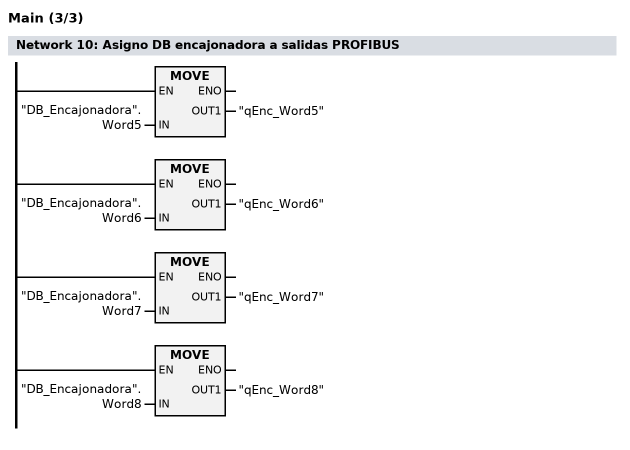
   RUNG wire#powerrail
      Move(in := "DB_Encajonadora".Word5, out1 => "qEnc_Word5")
   END_RUNG
   RUNG wire#powerrail
      Move(in := "DB_Encajonadora".Word6, out1 => "qEnc_Word6")
   END_RUNG
   RUNG wire#powerrail
      Move(in := "DB_Encajonadora".Word7, out1 => "qEnc_Word7")
   END_RUNG
   RUNG wire#powerrail
      Move(in := "DB_Encajonadora".Word8, out1 => "qEnc_Word8")
   END_RUNG
   // the same network as SCL:
   "qEnc_Word5" := "DB_Encajonadora".Word5;
   "qEnc_Word6" := "DB_Encajonadora".Word6;
   "qEnc_Word7" := "DB_Encajonadora".Word7;
   "qEnc_Word8" := "DB_Encajonadora".Word8;
END_REGION
END_ORGANIZATION_BLOCK

ORGANIZATION_BLOCK "Cyclic interrupt"   // OB30, LAD, CyclicInterrupt
{ S7_Optimized_Access := 'TRUE' }
VERSION : 0.1
   VAR_INPUT
      Initial_Call : Bool;   // Initial call of this OB
      Event_Count : Int;   // Events discarded
   END_VAR
BEGIN

REGION Network 1: Move
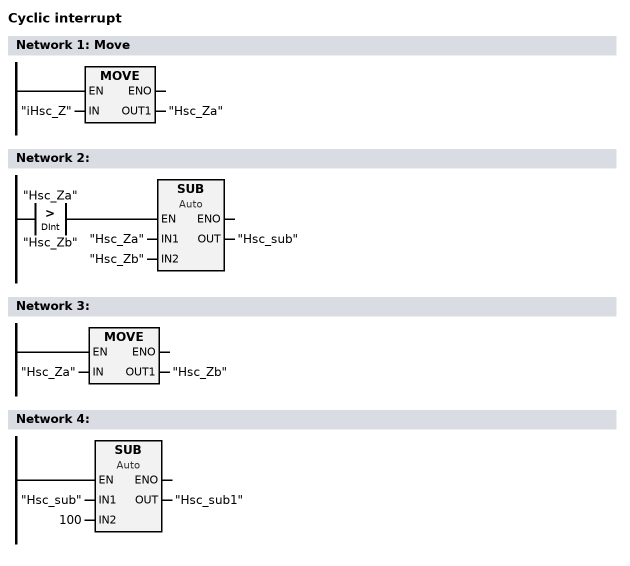
   RUNG wire#powerrail
      Move(in := "iHsc_Z", out1 => "Hsc_Za")
   END_RUNG
   // the same network as SCL:
   "Hsc_Za" := "iHsc_Z";
END_REGION

REGION Network 2
   RUNG wire#powerrail
      { S7_Templates := "SrcType := DInt" } GT_Contact(in1 := "Hsc_Za", in2 := "Hsc_Zb")
      Sub(in1 := "Hsc_Za", in2 := "Hsc_Zb", out => "Hsc_sub")
   END_RUNG
   // the same network as SCL:
   IF "Hsc_Za" > "Hsc_Zb" THEN "Hsc_sub" := "Hsc_Za" - "Hsc_Zb"; END_IF;
END_REGION

REGION Network 3
   RUNG wire#powerrail
      Move(in := "Hsc_Za", out1 => "Hsc_Zb")
   END_RUNG
   // the same network as SCL:
   "Hsc_Zb" := "Hsc_Za";
END_REGION

REGION Network 4
   RUNG wire#powerrail
      Sub(in1 := "Hsc_sub", in2 := 100, out => "Hsc_sub1")
   END_RUNG
   // the same network as SCL:
   "Hsc_sub1" := "Hsc_sub" - 100;
END_REGION
END_ORGANIZATION_BLOCK

// folder: ESTANDAR

FUNCTION_BLOCK "Motor M&CM"   // FB2, LAD
TITLE = Motor Marcha & Contra-Marcha
{ S7_Optimized_Access := 'TRUE' }
VERSION : 0.1
   VAR_INPUT
      iOrdMar_Dir : Bool;
      iOrdMar_Rev : Bool;
      iConfMar_Dir : Bool;
      iConfMar_Rev : Bool;
      iGMT : Bool;
      iTConf_Warn : Time;
      iTConf_Fall : Time;
      iTRearranque : Time;
   END_VAR
   VAR_OUTPUT
      oMar_Dir : Bool;
      oMar_Rev : Bool;
      oWarning_CTC_Dir : Bool;
      oWarning_CTC_Rev : Bool;
      oFall_CTC_Dir : Bool;
      oFall_CTC_Rev : Bool;
      oFall_GMT : Bool;
   END_VAR
   VAR
      IEC_Timer_0_Instance : IEC_TIMER;
      IEC_Timer_0_Instance_1 : IEC_TIMER;
      IEC_Timer_0_Instance_2 : IEC_TIMER;
      IEC_Timer_0_Instance_3 : IEC_TIMER;
      IEC_Timer_0_Instance_4 : IEC_TIMER;
      MarDir_Aux : Bool;
      MarRev_Aux : Bool;
   END_VAR
   VAR_TEMP
      Fall_GMT_Aux : Bool;
      Fall_CTC_Dir_Aux : Bool;
      Fall_CTC_Rev_Aux : Bool;
      Habil_Mov : Bool;
   END_VAR
   VAR_TEMP   // added for the SCL form of the ladder/FBD networks
      _w1 : Bool;
   END_VAR
BEGIN

REGION Network 1: Falla Guardamotor
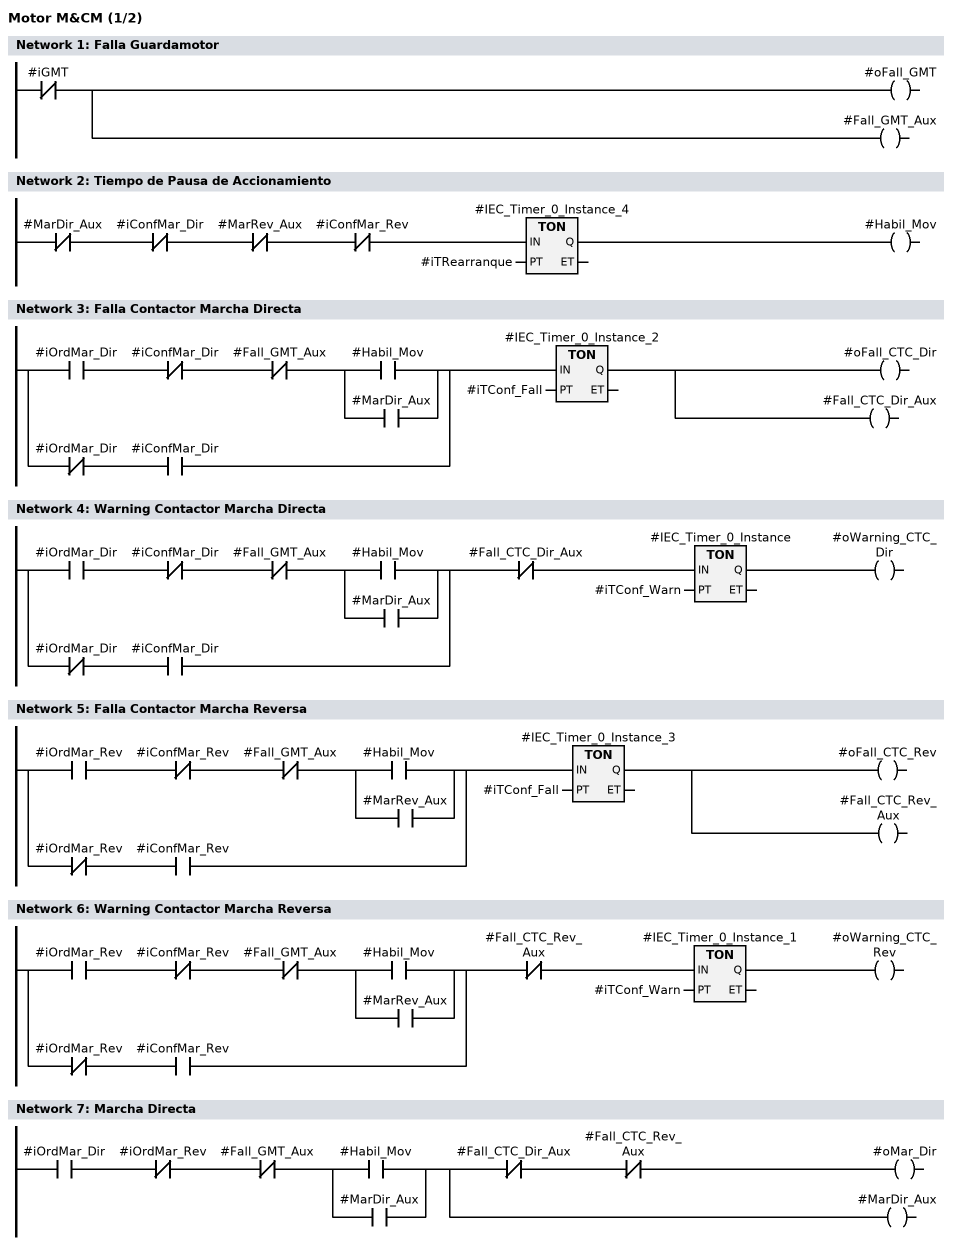
   RUNG wire#powerrail
      I_Contact( #iGMT )
      wire#w1
      Coil( #oFall_GMT )
   END_RUNG
   RUNG wire#w1
      Coil( #Fall_GMT_Aux )
   END_RUNG
   // the same network as SCL:
   #oFall_GMT := NOT #iGMT;
   #Fall_GMT_Aux := NOT #iGMT;
END_REGION

REGION Network 2: Tiempo de Pausa de Accionamiento
   #IEC_Timer_0_Instance_4.TON(IN := NOT #MarDir_Aux AND NOT #iConfMar_Dir AND NOT #MarRev_Aux AND NOT #iConfMar_Rev,
                           PT := #iTRearranque);
   #Habil_Mov := #IEC_Timer_0_Instance_4.Q;
END_REGION

REGION Network 3: Falla Contactor Marcha Directa
   #IEC_Timer_0_Instance_2.TON(IN := (#iOrdMar_Dir AND NOT #iConfMar_Dir AND NOT #Fall_GMT_Aux AND (#Habil_Mov OR #MarDir_Aux)) OR (NOT #iOrdMar_Dir AND #iConfMar_Dir),
                           PT := #iTConf_Fall);
   #oFall_CTC_Dir := #IEC_Timer_0_Instance_2.Q;
   #Fall_CTC_Dir_Aux := #IEC_Timer_0_Instance_2.Q;
END_REGION

REGION Network 4: Warning Contactor Marcha Directa
   #IEC_Timer_0_Instance.TON(IN := ((#iOrdMar_Dir AND NOT #iConfMar_Dir AND NOT #Fall_GMT_Aux AND (#Habil_Mov OR #MarDir_Aux)) OR (NOT #iOrdMar_Dir AND #iConfMar_Dir)) AND NOT #Fall_CTC_Dir_Aux,
                           PT := #iTConf_Warn);
   #oWarning_CTC_Dir := #IEC_Timer_0_Instance.Q;
END_REGION

REGION Network 5: Falla Contactor Marcha Reversa
   #IEC_Timer_0_Instance_3.TON(IN := (#iOrdMar_Rev AND NOT #iConfMar_Rev AND NOT #Fall_GMT_Aux AND (#Habil_Mov OR #MarRev_Aux)) OR (NOT #iOrdMar_Rev AND #iConfMar_Rev),
                           PT := #iTConf_Fall);
   #oFall_CTC_Rev := #IEC_Timer_0_Instance_3.Q;
   #Fall_CTC_Rev_Aux := #IEC_Timer_0_Instance_3.Q;
END_REGION

REGION Network 6: Warning Contactor Marcha Reversa
   #IEC_Timer_0_Instance_1.TON(IN := ((#iOrdMar_Rev AND NOT #iConfMar_Rev AND NOT #Fall_GMT_Aux AND (#Habil_Mov OR #MarRev_Aux)) OR (NOT #iOrdMar_Rev AND #iConfMar_Rev)) AND NOT #Fall_CTC_Rev_Aux,
                           PT := #iTConf_Warn);
   #oWarning_CTC_Rev := #IEC_Timer_0_Instance_1.Q;
END_REGION

REGION Network 7: Marcha Directa
   RUNG wire#powerrail
      Contact( #iOrdMar_Dir )
      I_Contact( #iOrdMar_Rev )
      I_Contact( #Fall_GMT_Aux )
      wire#w1
      Contact( #Habil_Mov )
      wire#w2
      I_Contact( #Fall_CTC_Dir_Aux )
      I_Contact( #Fall_CTC_Rev_Aux )
      Coil( #oMar_Dir )
   END_RUNG
   RUNG wire#w1
      Contact( #MarDir_Aux )
   END_RUNG wire#w2
   RUNG wire#w2
      Coil( #MarDir_Aux )
   END_RUNG
   // the same network as SCL:
   #_w1 := #iOrdMar_Dir AND NOT #iOrdMar_Rev AND NOT #Fall_GMT_Aux AND (#Habil_Mov OR #MarDir_Aux);
   #oMar_Dir := #_w1 AND NOT #Fall_CTC_Dir_Aux AND NOT #Fall_CTC_Rev_Aux;
   #MarDir_Aux := #_w1;
END_REGION

REGION Network 8: Marcha Reversa
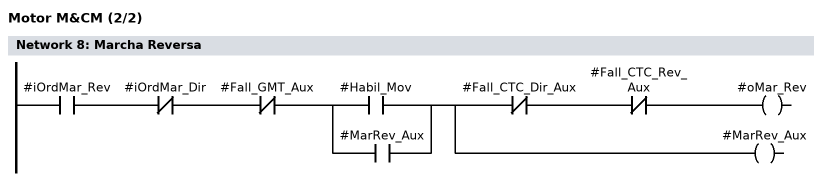
   RUNG wire#powerrail
      Contact( #iOrdMar_Rev )
      I_Contact( #iOrdMar_Dir )
      I_Contact( #Fall_GMT_Aux )
      wire#w1
      Contact( #Habil_Mov )
      wire#w2
      I_Contact( #Fall_CTC_Dir_Aux )
      I_Contact( #Fall_CTC_Rev_Aux )
      Coil( #oMar_Rev )
   END_RUNG
   RUNG wire#w1
      Contact( #MarRev_Aux )
   END_RUNG wire#w2
   RUNG wire#w2
      Coil( #MarRev_Aux )
   END_RUNG
   // the same network as SCL:
   #_w1 := #iOrdMar_Rev AND NOT #iOrdMar_Dir AND NOT #Fall_GMT_Aux AND (#Habil_Mov OR #MarRev_Aux);
   #oMar_Rev := #_w1 AND NOT #Fall_CTC_Dir_Aux AND NOT #Fall_CTC_Rev_Aux;
   #MarRev_Aux := #_w1;
END_REGION
END_FUNCTION_BLOCK

FUNCTION_BLOCK "FB_VAR_MOT"   // FB4, LAD
{ S7_Optimized_Access := 'FALSE' }
VERSION : 0.1
   VAR_INPUT
      "CMD Mar Dir" : Bool;   // Comando Marcha Directa
      "CMD Mar Rev" : Bool;   // Comando Marcha Reversa
      "HAB  Mar" : Bool;   // Habilita Marcha
      "SP Vel" : Real;   // Setpoint de Velocidad
      Reset : Bool;   // Comando resetear falla
      Fault : Bool;   // Indica variador en falla
      Ready : Bool;   // Indica variador Ready
      Ton_Freno : Time := T#400ms;
      Ton_Mar : Time := T#100ms;
      Tof_Freno : Time := T#100ms;
      Tof_Mar : Time := T#200ms;
   END_VAR
   VAR_OUTPUT
      Marcha : Bool;   // Orden de marcha a variador
      "Inv Giro" : Bool;   // Orden de invertir sentido de giro a variador
      "Reset Fault" : Bool;   // Reset Fault a variador
      Velocidad : Word;   // Referencia de Velocidad a variador
      Freno : Bool;   // Apertura de Freno
      Falla : Bool;   // Indica falla del variador
      Warning : Bool;   // Indica variador no Ready
   END_VAR
   VAR
      IEC_Timer_Freno : TON_TIME;
      IEC_Timer_Motor : TON_TIME;
      IEC_Timer_Reset : TOF_TIME;
      "_CMD Marcha Dir" : Bool;
      "_CMD Marcha Rev" : Bool;
      _CMD_AbrirFreno : Bool;
      IEC_Timer_0_Instance : TON_TIME;
      IEC_Timer_0_Instance_1 : TOF_TIME;
      IEC_Timer_0_Instance_2 : TOF_TIME;
      Ord_Marcha : Bool;
      Mem_Inv : Bool;
   END_VAR
   VAR_TEMP
      Vel_Real : Real;
      Vel_Int : Int;
      _Hab_Abrir_Freno : Bool;
      "Pre Marcha" : Bool;
      Aux : Bool;
      Freno_Aux : Bool;
   END_VAR
   VAR_TEMP   // added for the SCL form of the ladder/FBD networks
      _w1 : Bool;
      _w2 : Bool;
      _w3 : Bool;
   END_VAR
BEGIN

REGION Network 1: #Aux
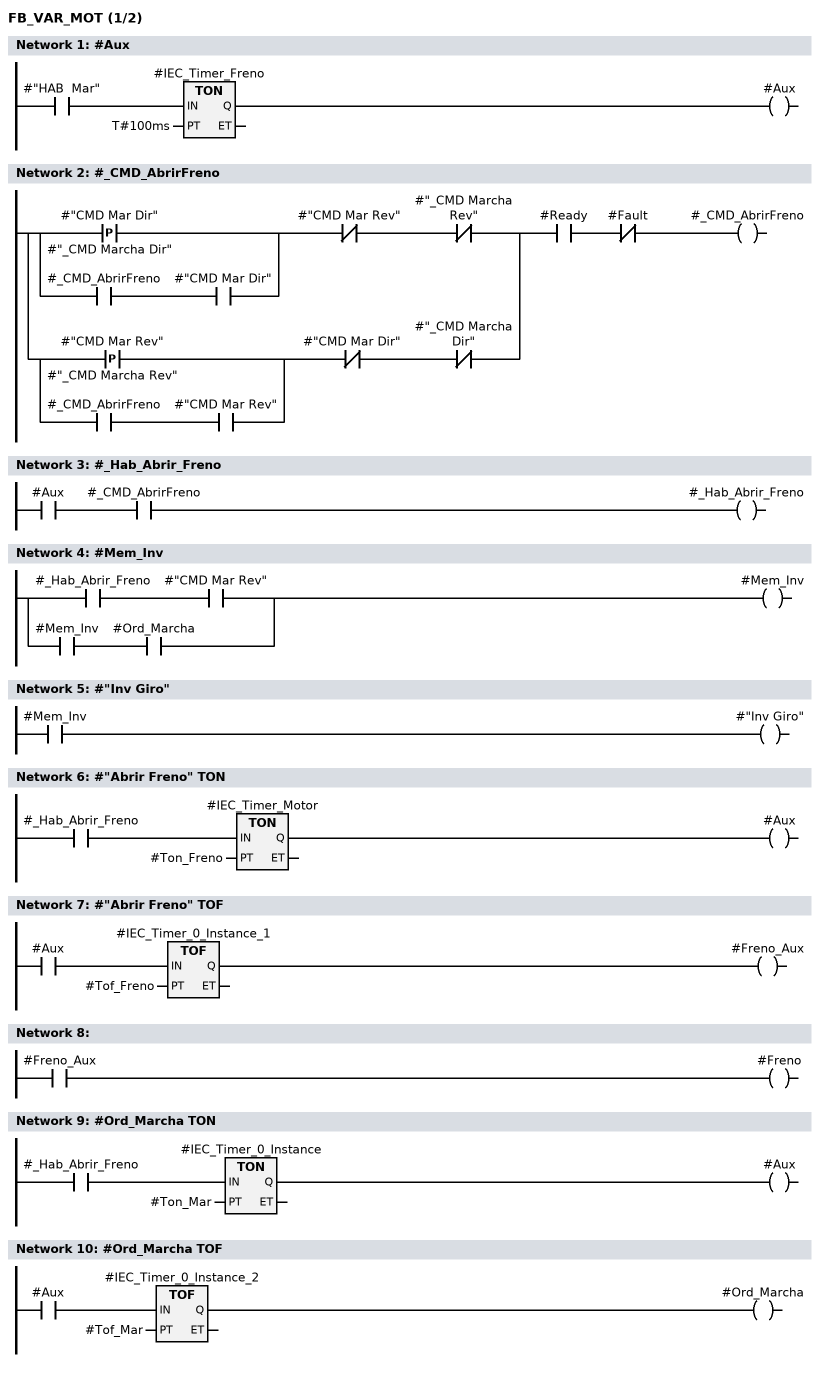
   #IEC_Timer_Freno(IN := #"HAB  Mar", PT := T#100ms);   // TON
   #Aux := #IEC_Timer_Freno.Q;
END_REGION

REGION Network 2: #_CMD_AbrirFreno
   RUNG wire#powerrail
      P_Contact(operand := #"CMD Mar Dir", bit := #"_CMD Marcha Dir")
      wire#w1
      I_Contact( #"CMD Mar Rev" )
      I_Contact( #"_CMD Marcha Rev" )
      wire#w2
      Contact( #Ready )
      I_Contact( #Fault )
      Coil( #_CMD_AbrirFreno )
   END_RUNG
   RUNG wire#powerrail
      Contact( #_CMD_AbrirFreno )
      Contact( #"CMD Mar Dir" )
   END_RUNG wire#w1
   RUNG wire#powerrail
      P_Contact(operand := #"CMD Mar Rev", bit := #"_CMD Marcha Rev")
      wire#w3
      I_Contact( #"CMD Mar Dir" )
      I_Contact( #"_CMD Marcha Dir" )
   END_RUNG wire#w2
   RUNG wire#powerrail
      Contact( #_CMD_AbrirFreno )
      Contact( #"CMD Mar Rev" )
   END_RUNG wire#w3
   // the same network as SCL:
   #_w1 := #"CMD Mar Dir" AND NOT #"_CMD Marcha Dir";   // rising edge of #"CMD Mar Dir"
   #"_CMD Marcha Dir" := #"CMD Mar Dir";
   #_w3 := (#_w1 OR (#_CMD_AbrirFreno AND #"CMD Mar Dir")) AND NOT #"CMD Mar Rev" AND NOT #"_CMD Marcha Rev";
   #_w2 := #"CMD Mar Rev" AND NOT #"_CMD Marcha Rev";   // rising edge of #"CMD Mar Rev"
   #"_CMD Marcha Rev" := #"CMD Mar Rev";
   #_CMD_AbrirFreno := (#_w3 OR ((#_w2 OR (#_CMD_AbrirFreno AND #"CMD Mar Rev")) AND NOT #"CMD Mar Dir" AND NOT #"_CMD Marcha Dir")) AND #Ready AND NOT #Fault;
END_REGION

REGION Network 3: #_Hab_Abrir_Freno
   RUNG wire#powerrail
      Contact( #Aux )
      Contact( #_CMD_AbrirFreno )
      Coil( #_Hab_Abrir_Freno )
   END_RUNG
   // the same network as SCL:
   #_Hab_Abrir_Freno := #Aux AND #_CMD_AbrirFreno;
END_REGION

REGION Network 4: #Mem_Inv
   RUNG wire#powerrail
      Contact( #_Hab_Abrir_Freno )
      Contact( #"CMD Mar Rev" )
      wire#w1
      Coil( #Mem_Inv )
   END_RUNG
   RUNG wire#powerrail
      Contact( #Mem_Inv )
      Contact( #Ord_Marcha )
   END_RUNG wire#w1
   // the same network as SCL:
   #Mem_Inv := (#_Hab_Abrir_Freno AND #"CMD Mar Rev") OR (#Mem_Inv AND #Ord_Marcha);
END_REGION

REGION Network 5: #"Inv Giro"
   RUNG wire#powerrail
      Contact( #Mem_Inv )
      Coil( #"Inv Giro" )
   END_RUNG
   // the same network as SCL:
   #"Inv Giro" := #Mem_Inv;
END_REGION

REGION Network 6: #"Abrir Freno" TON
   #IEC_Timer_Motor(IN := #_Hab_Abrir_Freno, PT := #Ton_Freno);   // TON
   #Aux := #IEC_Timer_Motor.Q;
END_REGION

REGION Network 7: #"Abrir Freno" TOF
   #IEC_Timer_0_Instance_1(IN := #Aux, PT := #Tof_Freno);   // TOF
   #Freno_Aux := #IEC_Timer_0_Instance_1.Q;
END_REGION

REGION Network 8
   RUNG wire#powerrail
      Contact( #Freno_Aux )
      Coil( #Freno )
   END_RUNG
   // the same network as SCL:
   #Freno := #Freno_Aux;
END_REGION

REGION Network 9: #Ord_Marcha TON
   #IEC_Timer_0_Instance(IN := #_Hab_Abrir_Freno, PT := #Ton_Mar);   // TON
   #Aux := #IEC_Timer_0_Instance.Q;
END_REGION

REGION Network 10: #Ord_Marcha TOF
   #IEC_Timer_0_Instance_2(IN := #Aux, PT := #Tof_Mar);   // TOF
   #Ord_Marcha := #IEC_Timer_0_Instance_2.Q;
END_REGION

REGION Network 11: #Marcha
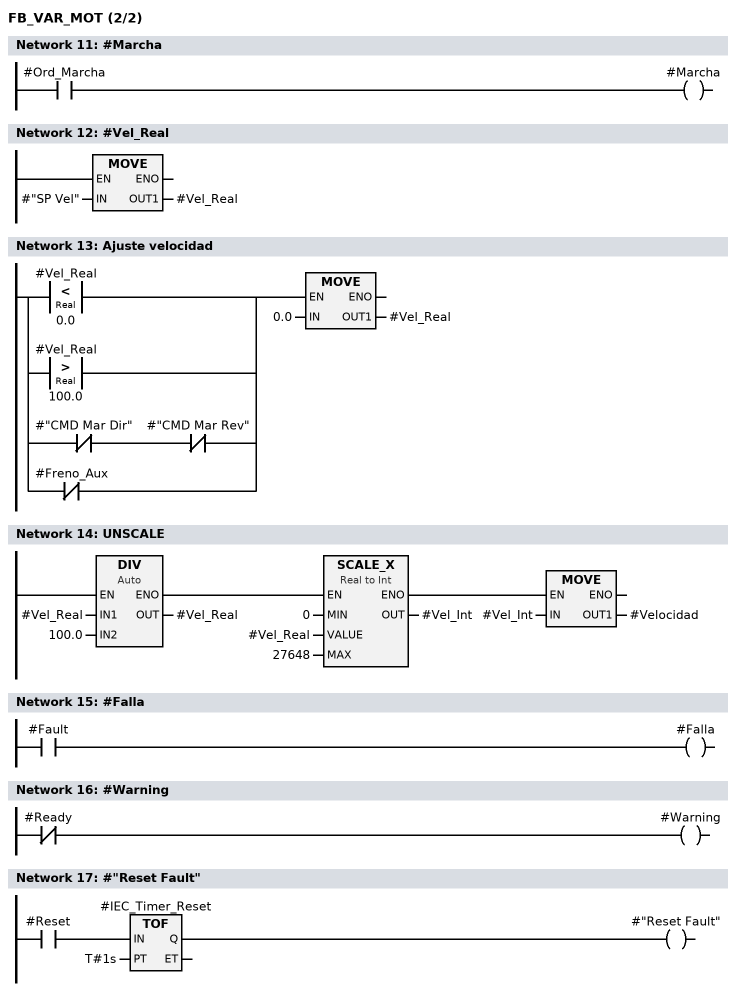
   RUNG wire#powerrail
      Contact( #Ord_Marcha )
      Coil( #Marcha )
   END_RUNG
   // the same network as SCL:
   #Marcha := #Ord_Marcha;
END_REGION

REGION Network 12: #Vel_Real
   RUNG wire#powerrail
      { S7_GenerateENO := "TRUE" } Move(in := #"SP Vel", out1 => #Vel_Real)
   END_RUNG
   // the same network as SCL:
   #Vel_Real := #"SP Vel";
END_REGION

REGION Network 13: Ajuste velocidad
   RUNG wire#powerrail
      { S7_Templates := "SrcType := Real" } LT_Contact(in1 := #Vel_Real, in2 := 0.0)
      wire#w1
      { S7_GenerateENO := "TRUE" } Move(in := 0.0, out1 => #Vel_Real)
   END_RUNG
   RUNG wire#powerrail
      { S7_Templates := "SrcType := Real" } GT_Contact(in1 := #Vel_Real, in2 := 100.0)
   END_RUNG wire#w1
   RUNG wire#powerrail
      I_Contact( #"CMD Mar Dir" )
      I_Contact( #"CMD Mar Rev" )
   END_RUNG wire#w1
   RUNG wire#powerrail
      I_Contact( #Freno_Aux )
   END_RUNG wire#w1
   // the same network as SCL:
   IF (#Vel_Real < 0.0) OR (#Vel_Real > 100.0) OR (NOT #"CMD Mar Dir" AND NOT #"CMD Mar Rev") OR NOT #Freno_Aux THEN
       #Vel_Real := 0.0;
   END_IF;
END_REGION

REGION Network 14: UNSCALE
   RUNG wire#powerrail
      Div(in1 := #Vel_Real, in2 := 100.0, out => #Vel_Real)
      { S7_Templates := "[SrcType := Real, DestType := Int]" } Scale(min := 0, value := #Vel_Real, max := 27648, out => #Vel_Int)
      { S7_GenerateENO := "TRUE" } Move(in := #Vel_Int, out1 => #Velocidad)
   END_RUNG
   // the same network as SCL:
   #Vel_Real := #Vel_Real / 100.0;
   #Vel_Int := SCALE_X(MIN := 0, VALUE := #Vel_Real, MAX := 27648);
   #Velocidad := #Vel_Int;
END_REGION

REGION Network 15: #Falla
   RUNG wire#powerrail
      Contact( #Fault )
      Coil( #Falla )
   END_RUNG
   // the same network as SCL:
   #Falla := #Fault;
END_REGION

REGION Network 16: #Warning
   RUNG wire#powerrail
      I_Contact( #Ready )
      Coil( #Warning )
   END_RUNG
   // the same network as SCL:
   #Warning := NOT #Ready;
END_REGION

REGION Network 17: #"Reset Fault"
   #IEC_Timer_Reset(IN := #Reset, PT := T#1s);   // TOF
   #"Reset Fault" := #IEC_Timer_Reset.Q;
END_REGION
END_FUNCTION_BLOCK

FUNCTION_BLOCK "Motor Simple"   // FB5, LAD
{ S7_Optimized_Access := 'TRUE' }
VERSION : 0.1
   VAR_INPUT
      iOrdMar : Bool;
      iConfMar : Bool;
      iGMT : Bool;
      iTConf_Warn : Time;
      iTConf_Fall : Time;
      iTRearranque : Time;
   END_VAR
   VAR_OUTPUT
      oMarcha : Bool;
      oWarning_CTC : Bool;
      oFall_CTC : Bool;
      oFall_GMT : Bool;
   END_VAR
   VAR
      IEC_Timer_0_Instance : IEC_TIMER;
      IEC_Timer_0_Instance_1 : IEC_TIMER;
      IEC_Timer_0_Instance_2 : IEC_TIMER;
      Mar_Aux : Bool;
   END_VAR
   VAR_TEMP
      Fall_GMT_Aux : Bool;
      Fall_CTC_Aux : Bool;
      Habil_Mov : Bool;
   END_VAR
BEGIN

REGION Network 1: Falla Guardamotor
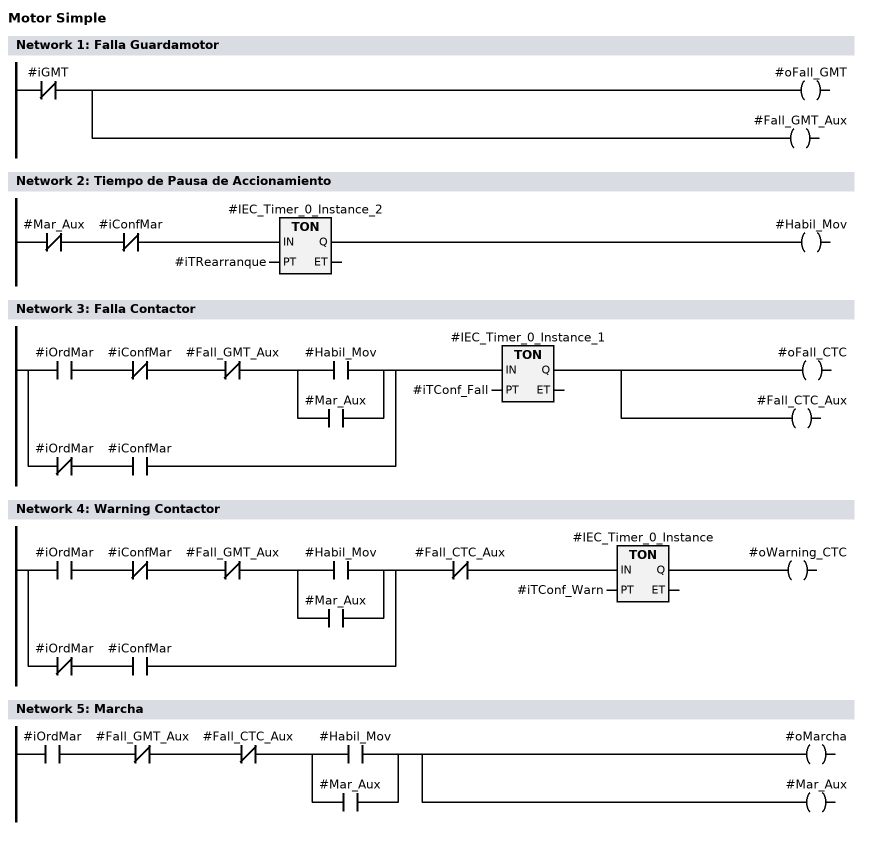
   RUNG wire#powerrail
      I_Contact( #iGMT )
      wire#w1
      Coil( #oFall_GMT )
   END_RUNG
   RUNG wire#w1
      Coil( #Fall_GMT_Aux )
   END_RUNG
   // the same network as SCL:
   #oFall_GMT := NOT #iGMT;
   #Fall_GMT_Aux := NOT #iGMT;
END_REGION

REGION Network 2: Tiempo de Pausa de Accionamiento
   #IEC_Timer_0_Instance_2.TON(IN := NOT #Mar_Aux AND NOT #iConfMar, PT := #iTRearranque);
   #Habil_Mov := #IEC_Timer_0_Instance_2.Q;
END_REGION

REGION Network 3: Falla Contactor
   #IEC_Timer_0_Instance_1.TON(IN := (#iOrdMar AND NOT #iConfMar AND NOT #Fall_GMT_Aux AND (#Habil_Mov OR #Mar_Aux)) OR (NOT #iOrdMar AND #iConfMar),
                           PT := #iTConf_Fall);
   #oFall_CTC := #IEC_Timer_0_Instance_1.Q;
   #Fall_CTC_Aux := #IEC_Timer_0_Instance_1.Q;
END_REGION

REGION Network 4: Warning Contactor
   #IEC_Timer_0_Instance.TON(IN := ((#iOrdMar AND NOT #iConfMar AND NOT #Fall_GMT_Aux AND (#Habil_Mov OR #Mar_Aux)) OR (NOT #iOrdMar AND #iConfMar)) AND NOT #Fall_CTC_Aux,
                           PT := #iTConf_Warn);
   #oWarning_CTC := #IEC_Timer_0_Instance.Q;
END_REGION

REGION Network 5: Marcha
   RUNG wire#powerrail
      Contact( #iOrdMar )
      I_Contact( #Fall_GMT_Aux )
      I_Contact( #Fall_CTC_Aux )
      wire#w1
      Contact( #Habil_Mov )
      wire#w2
      Coil( #oMarcha )
   END_RUNG
   RUNG wire#w1
      Contact( #Mar_Aux )
   END_RUNG wire#w2
   RUNG wire#w2
      Coil( #Mar_Aux )
   END_RUNG
   // the same network as SCL:
   #oMarcha := #iOrdMar AND NOT #Fall_GMT_Aux AND NOT #Fall_CTC_Aux AND (#Habil_Mov OR #Mar_Aux);
   #Mar_Aux := #oMarcha;
END_REGION
END_FUNCTION_BLOCK

FUNCTION_BLOCK "FB_VLV_2_POS"   // FB6, LAD
{ S7_Optimized_Access := 'FALSE' }
VERSION : 0.1
   VAR_INPUT
      Ir_Pos_1 : Bool;   // Comando Mover Cilindro a Posición 1, activar constantemente
      Ir_Pos_2 : Bool;   // Comando Mover Cilindro a Posición 2, activar constantemente
      Conf_Pos_1 : Bool;   // Confirmación Cilindro en Posición 1
      Conf_Pos_2 : Bool;   // Confirmación Cilindro en Posición 2
      T_Conf : Time := T#10s;   // Tiempo admisible para confirmación de posición
      T_ON : Time;   // Duración accionamiento salida [0 = constantemente]
   END_VAR
   VAR_OUTPUT
      Pos_1 : Bool;   // Orden Mover Cilindro a Posición 1
      Pos_2 : Bool;   // Orden Mover Cilindro a Posición 2
      ERROR : Int;   // 0 = Sin Error, 1 = Error Programación, 2 = Error Doble Confirmación, 3 = Error Confirmación Pos_1, 4 = Error Confirmación Pos_2, 5 = Sin Confirmaciones
   END_VAR
   VAR
      IEC_Timer_0_Instance : IEC_TIMER;
      IEC_Timer_0_Instance_1 : IEC_TIMER;
      IEC_Timer_0_Instance_2 : IEC_TIMER;
      IEC_Timer_0_Instance_3 : IEC_TIMER;
      IEC_Timer_0_Instance_4 : IEC_TIMER;
   END_VAR
   VAR_TEMP
      Aux_1 : Bool;   // Auxiliar 1
      Aux_2 : Bool;   // Auxiliar 2
      Aux_ERROR : Int;   // Auxiliar ERROR
   END_VAR
BEGIN

REGION Network 1: Auxiliar 1
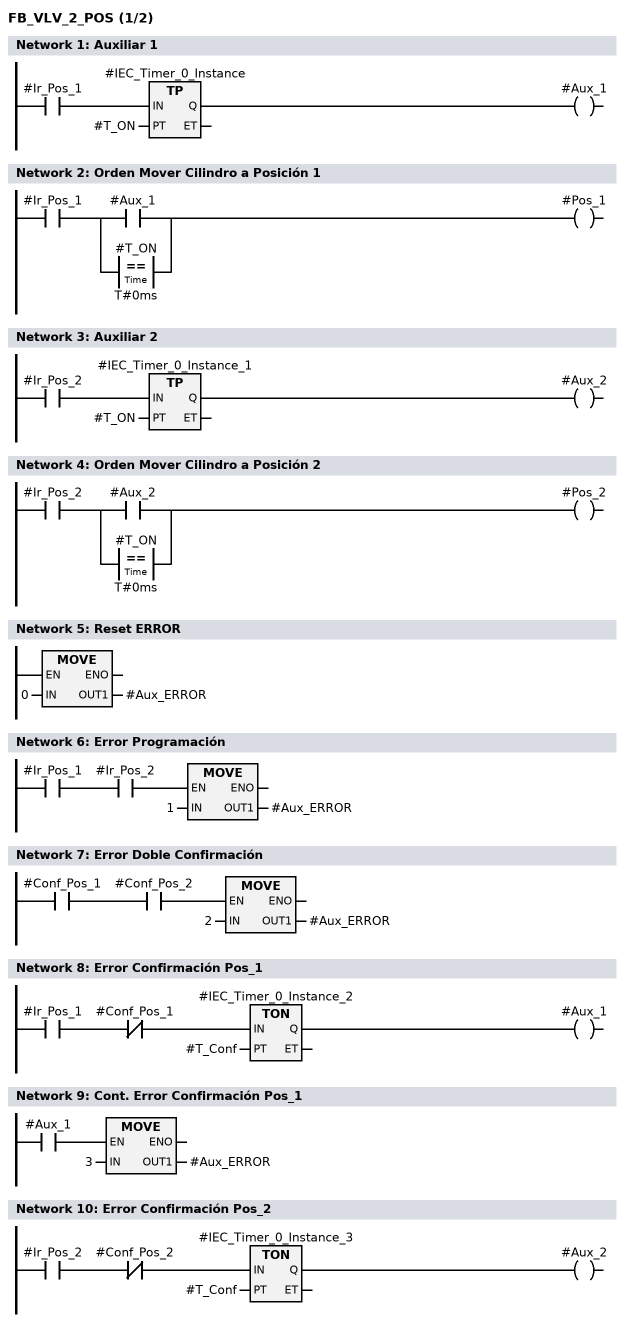
   #IEC_Timer_0_Instance.TP(IN := #Ir_Pos_1, PT := #T_ON);
   #Aux_1 := #IEC_Timer_0_Instance.Q;
END_REGION

REGION Network 2: Orden Mover Cilindro a Posición 1
   RUNG wire#powerrail
      Contact( #Ir_Pos_1 )
      wire#w1
      Contact( #Aux_1 )
      wire#w2
      Coil( #Pos_1 )
   END_RUNG
   RUNG wire#w1
      { S7_Templates := "SrcType := Time" } EQ_Contact(in1 := #T_ON, in2 := T#0ms)
   END_RUNG wire#w2
   // the same network as SCL:
   #Pos_1 := #Ir_Pos_1 AND (#Aux_1 OR (#T_ON = T#0ms));
END_REGION

REGION Network 3: Auxiliar 2
   #IEC_Timer_0_Instance_1.TP(IN := #Ir_Pos_2, PT := #T_ON);
   #Aux_2 := #IEC_Timer_0_Instance_1.Q;
END_REGION

REGION Network 4: Orden Mover Cilindro a Posición 2
   RUNG wire#powerrail
      Contact( #Ir_Pos_2 )
      wire#w1
      Contact( #Aux_2 )
      wire#w2
      Coil( #Pos_2 )
   END_RUNG
   RUNG wire#w1
      { S7_Templates := "SrcType := Time" } EQ_Contact(in1 := #T_ON, in2 := T#0ms)
   END_RUNG wire#w2
   // the same network as SCL:
   #Pos_2 := #Ir_Pos_2 AND (#Aux_2 OR (#T_ON = T#0ms));
END_REGION

REGION Network 5: Reset ERROR
   RUNG wire#powerrail
      { S7_GenerateENO := "TRUE" } Move(in := 0, out1 => #Aux_ERROR)
   END_RUNG
   // the same network as SCL:
   #Aux_ERROR := 0;
END_REGION

REGION Network 6: Error Programación
   RUNG wire#powerrail
      Contact( #Ir_Pos_1 )
      Contact( #Ir_Pos_2 )
      { S7_GenerateENO := "TRUE" } Move(in := 1, out1 => #Aux_ERROR)
   END_RUNG
   // the same network as SCL:
   IF #Ir_Pos_1 AND #Ir_Pos_2 THEN #Aux_ERROR := 1; END_IF;
END_REGION

REGION Network 7: Error Doble Confirmación
   RUNG wire#powerrail
      Contact( #Conf_Pos_1 )
      Contact( #Conf_Pos_2 )
      { S7_GenerateENO := "TRUE" } Move(in := 2, out1 => #Aux_ERROR)
   END_RUNG
   // the same network as SCL:
   IF #Conf_Pos_1 AND #Conf_Pos_2 THEN #Aux_ERROR := 2; END_IF;
END_REGION

REGION Network 8: Error Confirmación Pos_1
   #IEC_Timer_0_Instance_2.TON(IN := #Ir_Pos_1 AND NOT #Conf_Pos_1, PT := #T_Conf);
   #Aux_1 := #IEC_Timer_0_Instance_2.Q;
END_REGION

REGION Network 9: Cont. Error Confirmación Pos_1
   RUNG wire#powerrail
      Contact( #Aux_1 )
      { S7_GenerateENO := "TRUE" } Move(in := 3, out1 => #Aux_ERROR)
   END_RUNG
   // the same network as SCL:
   IF #Aux_1 THEN #Aux_ERROR := 3; END_IF;
END_REGION

REGION Network 10: Error Confirmación Pos_2
   #IEC_Timer_0_Instance_3.TON(IN := #Ir_Pos_2 AND NOT #Conf_Pos_2, PT := #T_Conf);
   #Aux_2 := #IEC_Timer_0_Instance_3.Q;
END_REGION

REGION Network 11: Cont. Error Confirmación Pos_2
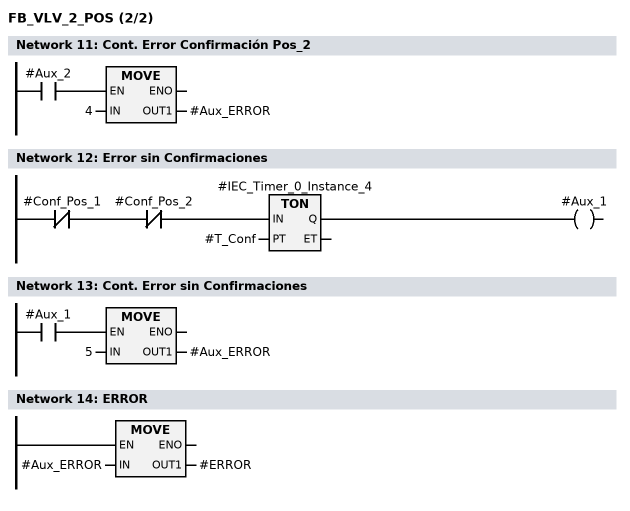
   RUNG wire#powerrail
      Contact( #Aux_2 )
      { S7_GenerateENO := "TRUE" } Move(in := 4, out1 => #Aux_ERROR)
   END_RUNG
   // the same network as SCL:
   IF #Aux_2 THEN #Aux_ERROR := 4; END_IF;
END_REGION

REGION Network 12: Error sin Confirmaciones
   #IEC_Timer_0_Instance_4.TON(IN := NOT #Conf_Pos_1 AND NOT #Conf_Pos_2, PT := #T_Conf);
   #Aux_1 := #IEC_Timer_0_Instance_4.Q;
END_REGION

REGION Network 13: Cont. Error sin Confirmaciones
   RUNG wire#powerrail
      Contact( #Aux_1 )
      { S7_GenerateENO := "TRUE" } Move(in := 5, out1 => #Aux_ERROR)
   END_RUNG
   // the same network as SCL:
   IF #Aux_1 THEN #Aux_ERROR := 5; END_IF;
END_REGION

REGION Network 14: ERROR
   RUNG wire#powerrail
      { S7_GenerateENO := "TRUE" } Move(in := #Aux_ERROR, out1 => #ERROR)
   END_RUNG
   // the same network as SCL:
   #ERROR := #Aux_ERROR;
END_REGION
END_FUNCTION_BLOCK

FUNCTION "MAQ_EST_32" : Void   // FC7, SCL
TITLE = Máquina de Estados 32
{ S7_Optimized_Access := 'TRUE' }
AUTHOR : FRD
FAMILY : MTA
NAME : MaqEst32
VERSION : 1.0
// KNOW_HOW_PROTECT  Máquina de estados de hasta 32 estados.
   VAR_INPUT
      Concatenadoras : DWord;   // Próximo estado de transición normal
      Prioritarias : DWord;   // Próximo estado de transición forzada
   END_VAR
   VAR_OUTPUT
      Error_Concatenadoras : Bool;   // Error en la programación de las Concatenadoras
      Error_Prioritarias : Bool;   // Error en la programación de las Prioritarias
   END_VAR
   VAR_IN_OUT
      Estado : DWord;   // Estado actual
   END_VAR
   VAR_TEMP
      Concat_Int : Int;   // Auxiliar INT para verificar las Concatenadoras
      Priorit_Int : Int;   // Auxiliar INT para verificar las Prioritarias
      Concat_Dword : DWord;   // Auxiliar DWORD para verificar las Concatenadoras
      Priorit_Dword : DWord;   // Auxiliar DWORD para verificar las Prioritarias
      Activar_Concat : Bool;   // Bit que indica Concatenadoras correctas
      Activar_Priorit : Bool;   // Bit que indica Prioritarias correctas
      Falla_Concat : Bool;   // Bit que indica falla en Concatenadoras
      Falla_Priorit : Bool;   // Bit que indica falla en Prioritarias
   END_VAR
BEGIN
   #Falla_Concat := 0;
   #Activar_Concat := 0;
   #Falla_Priorit := 0;
   #Activar_Priorit := 0; 
   #Error_Concatenadoras := 0;
   #Error_Prioritarias := 0;

   IF #Concatenadoras <> 0 THEN     //Evaluar Concatenadoras si son distintas de "0"

    #Concat_Int := ENCO(IN := #Concatenadoras );  //Convierte posición_DWORD en INT (0 a 31), lee el LSb

    #Concat_Dword := DECO(IN := INT_TO_UINT(#Concat_Int));//Convierte INT en posición_DWORD (1 a 32)

    IF #Concatenadoras = #Concat_Dword THEN  //Si son iguales, había sólo un bit en "1"

     #Activar_Concat := 1;    //Concatenadora correcta

    ELSE

     #Falla_Concat := 1;    //Falla en Concatenadora

    END_IF;

   END_IF;

   IF #Prioritarias <> 0 THEN     //Evaluar Prioritarias si son distintas de "0"

    #Priorit_Int := ENCO(IN := #Prioritarias);  //Convierte posición_DWORD en INT (0 a 31), lee el LSb

    #Priorit_Dword := DECO(IN := INT_TO_UINT(#Priorit_Int));//Convierte INT en posición_DWORD (1 a 32)

    IF #Prioritarias = #Priorit_Dword THEN  //Si son iguales, había sólo un bit en "1"

     #Activar_Priorit := 1;   //Prioritaria correcta

    ELSE

     #Falla_Priorit := 1;    //Falla en Prioritaria

    END_IF;

   END_IF;

   IF NOT(#Falla_Priorit OR #Falla_Concat) THEN  //Si no hay falla de Prioritaria ni de Concatenadora

    IF #Activar_Priorit THEN    //Si hay que asignar Prioritarias

     #Estado := #Prioritarias;

    ELSE

     IF #Activar_Concat THEN   //Si hay que asignar Concatenadoras

      #Estado := #Concatenadoras;

     END_IF;

    END_IF;

   ELSE

    IF #Falla_Concat THEN     //Si hay falla de Concatenadoras

     #Error_Concatenadoras := 1;    //Activar Error_Concatenadoras

    END_IF;

    IF #Falla_Priorit THEN    //Si hay falla de Prioritarias

     #Error_Prioritarias := 1;    //Activar Error_Prioritarias

    END_IF;

   END_IF;
END_FUNCTION

// folder: INCIDENTES

FUNCTION_BLOCK "FB_INC_GENERAL"   // FB500, LAD
TITLE = ALARMAS GENERAL
{ S7_Optimized_Access := 'FALSE' }
VERSION : 0.1
   VAR
      Alarma_On : Bool;
   END_VAR
BEGIN

REGION Network 1: Alarma 0 - Protecciones abiertas
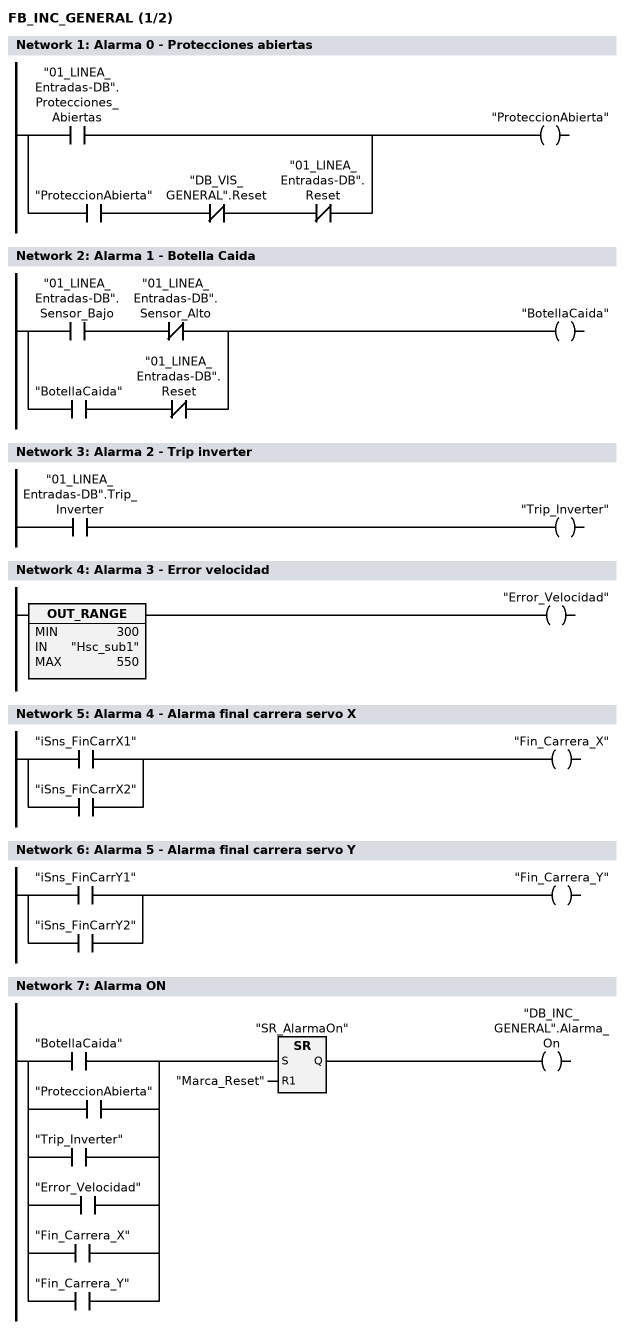
   RUNG wire#powerrail
      Contact( "01_LINEA_Entradas-DB".Protecciones_Abiertas )
      wire#w1
      Coil( "ProteccionAbierta" )
   END_RUNG
   RUNG wire#powerrail
      Contact( "ProteccionAbierta" )
      I_Contact( "DB_VIS_GENERAL".Reset )
      I_Contact( "01_LINEA_Entradas-DB".Reset )
   END_RUNG wire#w1
   // the same network as SCL:
   "ProteccionAbierta" := "01_LINEA_Entradas-DB".Protecciones_Abiertas OR ("ProteccionAbierta" AND NOT "DB_VIS_GENERAL".Reset AND NOT "01_LINEA_Entradas-DB".Reset);
END_REGION

REGION Network 2: Alarma 1 - Botella Caida
   RUNG wire#powerrail
      Contact( "01_LINEA_Entradas-DB".Sensor_Bajo )
      I_Contact( "01_LINEA_Entradas-DB".Sensor_Alto )
      wire#w1
      Coil( "BotellaCaida" )
   END_RUNG
   RUNG wire#powerrail
      Contact( "BotellaCaida" )
      I_Contact( "01_LINEA_Entradas-DB".Reset )
   END_RUNG wire#w1
   // the same network as SCL:
   "BotellaCaida" := ("01_LINEA_Entradas-DB".Sensor_Bajo AND NOT "01_LINEA_Entradas-DB".Sensor_Alto) OR ("BotellaCaida" AND NOT "01_LINEA_Entradas-DB".Reset);
END_REGION

REGION Network 3: Alarma 2 - Trip inverter
   RUNG wire#powerrail
      Contact( "01_LINEA_Entradas-DB".Trip_Inverter )
      Coil( "Trip_Inverter" )
   END_RUNG
   // the same network as SCL:
   "Trip_Inverter" := "01_LINEA_Entradas-DB".Trip_Inverter;
END_REGION

REGION Network 4: Alarma 3 - Error velocidad
   "Error_Velocidad" := ("Hsc_sub1" < 300) OR ("Hsc_sub1" > 550);
END_REGION

REGION Network 5: Alarma 4 - Alarma final carrera servo X
   RUNG wire#powerrail
      Contact( "iSns_FinCarrX1" )
      wire#w1
      Coil( "Fin_Carrera_X" )
   END_RUNG
   RUNG wire#powerrail
      Contact( "iSns_FinCarrX2" )
   END_RUNG wire#w1
   // the same network as SCL:
   "Fin_Carrera_X" := "iSns_FinCarrX1" OR "iSns_FinCarrX2";
END_REGION

REGION Network 6: Alarma 5 - Alarma final carrera servo Y
   RUNG wire#powerrail
      Contact( "iSns_FinCarrY1" )
      wire#w1
      Coil( "Fin_Carrera_Y" )
   END_RUNG
   RUNG wire#powerrail
      Contact( "iSns_FinCarrY2" )
   END_RUNG wire#w1
   // the same network as SCL:
   "Fin_Carrera_Y" := "iSns_FinCarrY1" OR "iSns_FinCarrY2";
END_REGION

REGION Network 7: Alarma ON
   RUNG wire#powerrail
      Contact( "BotellaCaida" )
      wire#w1
      S_SR(operand := "SR_AlarmaOn", r1 := "Marca_Reset")
      Coil( "DB_INC_GENERAL".Alarma_On )
   END_RUNG
   RUNG wire#powerrail
      Contact( "ProteccionAbierta" )
   END_RUNG wire#w1
   RUNG wire#powerrail
      Contact( "Trip_Inverter" )
   END_RUNG wire#w1
   RUNG wire#powerrail
      Contact( "Error_Velocidad" )
   END_RUNG wire#w1
   RUNG wire#powerrail
      Contact( "Fin_Carrera_X" )
   END_RUNG wire#w1
   RUNG wire#powerrail
      Contact( "Fin_Carrera_Y" )
   END_RUNG wire#w1
   // the same network as SCL:
   IF "BotellaCaida" OR "ProteccionAbierta" OR "Trip_Inverter" OR "Error_Velocidad" OR "Fin_Carrera_X" OR "Fin_Carrera_Y" THEN
       "SR_AlarmaOn" := TRUE;   // SR flip-flop
   END_IF;
   IF "Marca_Reset" THEN "SR_AlarmaOn" := FALSE; END_IF;
   "DB_INC_GENERAL".Alarma_On := "SR_AlarmaOn";
END_REGION

REGION Network 8: Encendido Semaforo Rojo
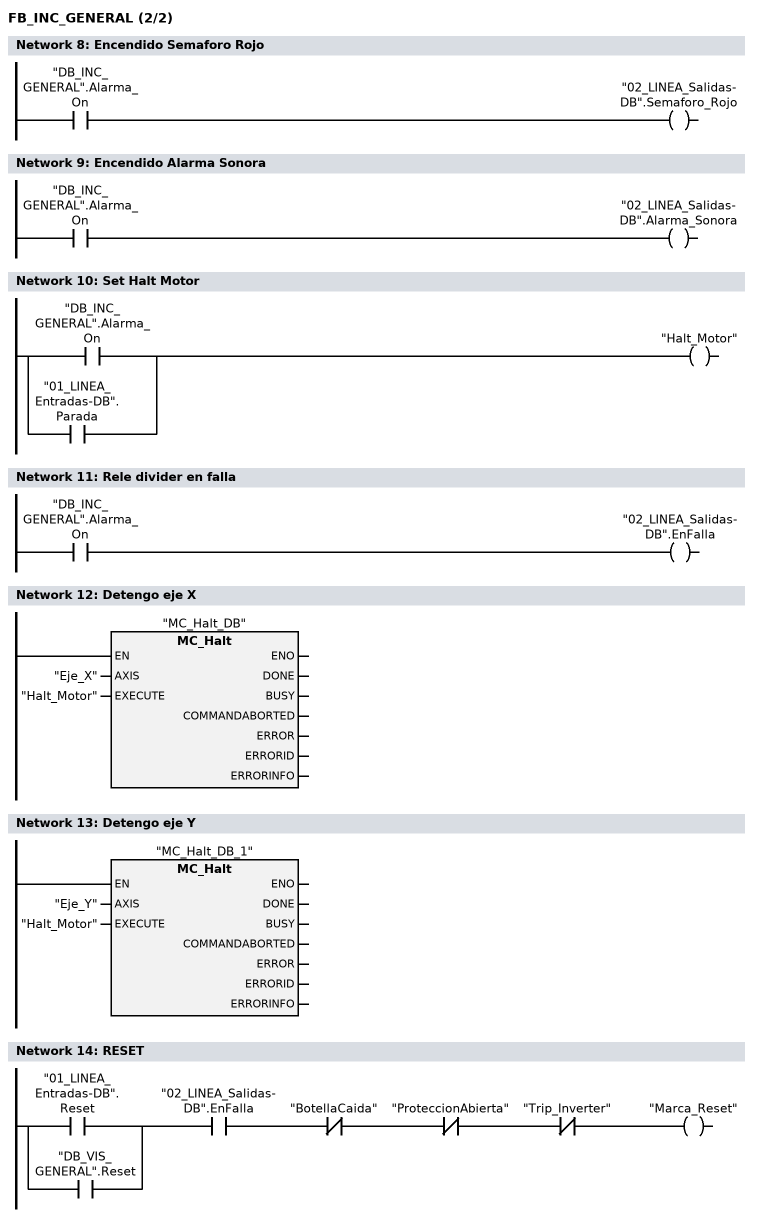
   RUNG wire#powerrail
      Contact( "DB_INC_GENERAL".Alarma_On )
      Coil( "02_LINEA_Salidas-DB".Semaforo_Rojo )
   END_RUNG
   // the same network as SCL:
   "02_LINEA_Salidas-DB".Semaforo_Rojo := "DB_INC_GENERAL".Alarma_On;
END_REGION

REGION Network 9: Encendido Alarma Sonora
   RUNG wire#powerrail
      Contact( "DB_INC_GENERAL".Alarma_On )
      Coil( "02_LINEA_Salidas-DB".Alarma_Sonora )
   END_RUNG
   // the same network as SCL:
   "02_LINEA_Salidas-DB".Alarma_Sonora := "DB_INC_GENERAL".Alarma_On;
END_REGION

REGION Network 10: Set Halt Motor
   RUNG wire#powerrail
      Contact( "DB_INC_GENERAL".Alarma_On )
      wire#w1
      Coil( "Halt_Motor" )
   END_RUNG
   RUNG wire#powerrail
      Contact( "01_LINEA_Entradas-DB".Parada )
   END_RUNG wire#w1
   // the same network as SCL:
   "Halt_Motor" := "DB_INC_GENERAL".Alarma_On OR "01_LINEA_Entradas-DB".Parada;
END_REGION

REGION Network 11: Rele divider en falla
   RUNG wire#powerrail
      Contact( "DB_INC_GENERAL".Alarma_On )
      Coil( "02_LINEA_Salidas-DB".EnFalla )
   END_RUNG
   // the same network as SCL:
   "02_LINEA_Salidas-DB".EnFalla := "DB_INC_GENERAL".Alarma_On;
END_REGION

REGION Network 12: Detengo eje X
   "MC_Halt_DB"(Axis := "Eje_X", Execute := "Halt_Motor");   // MC_Halt
END_REGION

REGION Network 13: Detengo eje Y
   "MC_Halt_DB_1"(Axis := "Eje_Y", Execute := "Halt_Motor");   // MC_Halt
END_REGION

REGION Network 14: RESET
   RUNG wire#powerrail
      Contact( "01_LINEA_Entradas-DB".Reset )
      wire#w1
      Contact( "02_LINEA_Salidas-DB".EnFalla )
      I_Contact( "BotellaCaida" )
      I_Contact( "ProteccionAbierta" )
      I_Contact( "Trip_Inverter" )
      Coil( "Marca_Reset" )
   END_RUNG
   RUNG wire#powerrail
      Contact( "DB_VIS_GENERAL".Reset )
   END_RUNG wire#w1
   // the same network as SCL:
   "Marca_Reset" := ("01_LINEA_Entradas-DB".Reset OR "DB_VIS_GENERAL".Reset) AND "02_LINEA_Salidas-DB".EnFalla AND NOT "BotellaCaida" AND NOT "ProteccionAbierta" AND NOT "Trip_Inverter";
END_REGION
END_FUNCTION_BLOCK

(* ===== HMI "HMI_RT_1" =====
system functions are stored by id; their names below are inferred from use
connection "Conexión_1": ETHERNET, SMART_S7_1200_OMS
connection "HMI_Conexión_1": ETHERNET, SMART_S7_1200_OMS

HMI tags "Tabla de variables estándar"
   "MC_Power_X" : Bool = PLC DB_VIS_GENERAL.MC_Pwr_EnX AT %DB800.DBX2.2, 1 s
   "MC_Power_Y" : Bool = PLC DB_VIS_GENERAL.MC_Pwrt_EnY AT %DB800.DBX2.3, 1 s
   "MC_JogFwd_X" : Bool = PLC DB_VIS_GENERAL.MC_JogFwd_X AT %DB800.DBX2.6, 1 s
   "MC_JogFwd_Y" : Bool = PLC DB_VIS_GENERAL.MC_JogFwd_Y AT %DB800.DBX2.7, 1 s
   "MC_JogBckWd_X" : Bool = PLC DB_VIS_GENERAL.MC_JogBwd_X AT %DB800.DBX3.0, 1 s
   "MC_JogBckWd_Y" : Bool = PLC DB_VIS_GENERAL.MC_JogBwd_Y AT %DB800.DBX3.1, 1 s
   "Falla_Divider" : Bool = PLC "02_LINEA_Salidas-DB".EnFalla AT %DB1.DBX0.0, 1 s
   "ProteccionesAbiertas" : Bool = PLC "01_LINEA_Entradas-DB".Protecciones_Abiertas AT %DB1.DBX0.0, 1 s
   "BotellaCaida" : Bool = PLC BotellaCaida AT %M100.1, 1 s
   "Marcha_Divider" : Bool = PLC "02_LINEA_Salidas-DB".EnMarcha AT %DB1.DBX0.0, 1 s
   "Trip_Inverter" : Bool = PLC Trip_Inverter AT %M100.2, 1 s
   "Cant_Bot" : Int = PLC DB_VIS_GENERAL.CantBot AT %DB800.DBW0, 1 s
   "Marcha" : Bool = PLC DB_VIS_GENERAL.Start AT %DB800.DBX3.4, 1 s
   "HomingOk" : Bool = PLC DB_VIS_GENERAL.HomingOk AT %DB800.DBX3.2, 1 s
   "Reset" : Bool = PLC DB_VIS_GENERAL.Reset AT %DB800.DBX3.3, 1 s
   "PM_MovX" : Real = PLC DB_PUESTA_MARCHA.MovXmm AT %DB1.DBX0.0, 1 s
   "PM_MovY" : Real = PLC DB_PUESTA_MARCHA.MovYmm AT %DB1.DBX0.0, 1 s
   "PM_TChFull" : Time = PLC DB_PUESTA_MARCHA.TChFull AT %DB1.DBX0.0, 1 s
   "Alarmas_1" : Word = PLC Alarmas_1 AT %MW100, 1 s
   "Alarma_ON" : Bool = PLC DB_INC_GENERAL.Alarma_On AT %DB500.DBX0.0, 1 s

discrete alarms
   1: 'Alarma 0 - Protecciones abiertas', class Errors, trigger "Alarmas_1" bit 8
   2: 'Alarma 1 - Botella caida', class Errors, trigger "Alarmas_1" bit 9
   3: 'Alarma 2 - Trip Inverter', class Errors, trigger "Alarmas_1" bit 10
   4: 'Alarma 3 - Error de velocidad', class Errors, trigger "Alarmas_1" bit 11
   5: 'Alarma 4 - Final de carrera X', class Errors, trigger "Alarmas_1" bit 12
   6: 'Alarma 5 - Final de carrera Y', class Errors, trigger "Alarmas_1" bit 13

text list "Cant_Bot": 0 '0'; 2 '2'; 4 '4'; 6 '6'; 8 '8'; 10 '10'; 12 '12'; 14 '14'; 16 '16'; 18 '18'; 20 '20'

text list "DesplazamientoX": 0 '0'; 60 '60'; 20 '20'; 40 '40'

screen "02 - Estado" 800x480, template "Plantilla_1"
   Button "Botón_2" at 162,433 size 160x47; TextOff 'Fallas'
      on Click: ActivateScreen("03 - Registro alarmas", 0)
      Appearance <- "Alarma_ON"
   TextField "Campo de texto_13" at 340,308 size 197x34; Text 'Divider en falla'
   GraphicIOField "PlotLight_Round_R_2" at 222,278 size 108x108; PictureOff "PilotLight_Round_R_Off_256c"; PictureOn "PilotLight_Round_R_On_256c"
      ProcessValue <- "Falla_Divider"
   GraphicIOField "PlotLight_Round_G_16" at 223,153 size 108x108; PictureOff "PilotLight_Round_G_Off_256c"; PictureOn "PilotLight_Round_G_On_256c"
      ProcessValue <- "Marcha_Divider"
   TextField "Campo de texto_14" at 340,187 size 235x34; Text 'Divider en marcha'
   Button "Botón_3" at 14,210 size 144x51; TextOff 'START'
      on Click: SetBit("Marcha")
   SymbolicIOField "Campo ES simbólico_1" at 222,81 size 104x49; TextOn '1'; TextOff '0'; TextList "Cant_Bot"
      ProcessValue <- "Cant_Bot"
   TextField "Campo de texto_2" at 340,87 size 385x34; Text 'Cantidad de botellas por carril'
   TextField "Campo de texto_1" at 10,406 size 148x17; Text 'Solo con Divider detenido'
   Button "Botón_4" at 640,431 size 159x48; TextOff 'Protegido'; Authorization "Administración de usuarios"
      on Click: ActivateScreen("04 - Puesta en marcha", 0)
   Button "Botón_1" at 1,433 size 161x47; TextOff 'Homing'
      on Click: ActivateScreen("01 - Pantalla_Inicializacion", 0)
      Visibility <- "Marcha"
   Button "Botón_5" at 2,433 size 161x47; TextOff 'Homing'
      Visibility <- "Marcha"

screen "01 - Pantalla_Inicializacion" 800x480, template "Plantilla_1"
   Button "Botón_1" at 321,433 size 161x47; TextOff 'HOMING OK'
      on Click: ActivateScreen("02 - Estado", 0); SetBit("HomingOk"); ResetBit("Reset")
   TextField "Campo de texto_1" at 49,36 size 704x94; Text '1. HABILITE AMBOS EJES 2. POSICIONE DIVIDER EN CARRIL 1 CON PULSADORES 3. PRESIONE HOMING OK UNA VEZ FINALIZADO'
   Button "FB_ArrowDown_Round" at 144,309 size 74x74; TextOff 'Text'; PictureOff "FB_ArrowDown_Round_Released_256c"; PictureOn "FB_ArrowDown_Round_Pressed_256c"
      on Release: ResetBit("MC_JogFwd_X")
      on Press: SetBit("MC_JogFwd_X")
   Button "FB_ArrowUp_Round" at 250,309 size 74x74; TextOff 'Text'; PictureOff "FB_ArrowUp_Round_Released_256c"; PictureOn "FB_ArrowUp_Round_Pressed_256c"
      on Release: ResetBit("MC_JogBckWd_X")
      on Press: SetBit("MC_JogBckWd_X")
   Button "FB_ArrowLeft_Round" at 488,308 size 74x74; TextOff 'Text'; PictureOff "FB_ArrowLeft_Round_Released_256c"; PictureOn "FB_ArrowLeft_Round_Pressed_256c"
      on Press: SetBit("MC_JogFwd_Y")
      on Release: ResetBit("MC_JogFwd_Y")
   Button "FB_ArrowRight_Round" at 594,309 size 74x74; TextOff 'Text'; PictureOff "FB_ArrowRight_Round_Released_256c"; PictureOn "FB_ArrowRight_Round_Pressed_256c"
      on Press: SetBit("MC_JogBckWd_Y")
      on Release: ResetBit("MC_JogBckWd_Y")
   Button "FB_Check_Round" at 199,199 size 74x74; TextOff 'Text'; PictureOn "FB_Check_Round_Pressed_256c"; PictureOff "FB_Check_Round_Released_256c"
      on Click: InvertBit("MC_Power_X")
      Appearance <- "MC_Power_X"
   Button "FB_Check_Round_1" at 544,199 size 74x74; TextOff 'Text'; PictureOff "FB_Check_Round_Released_256c"; PictureOn "FB_Check_Round_Pressed_256c"
      on Click: InvertBit("MC_Power_Y")
      Appearance <- "MC_Power_Y"
   TextField "Campo de texto_3" at 174,154 size 123x23; Text 'Habilitar eje X'
   TextField "Campo de texto_2" at 519,154 size 123x23; Text 'Habilitar eje Y'
   TextField "Campo de texto_4" at 372,177 size 16x23; Text 'Text'
   Button "Botón_2" at 162,433 size 160x47; TextOff 'Fallas'
      on Click: ActivateScreen("03 - Registro alarmas", 0)
      Appearance <- "Alarma_ON"
   Button "Botón_4" at 640,431 size 159x48; TextOff 'Protegido'; Authorization "Administración de usuarios"
      on Click: ActivateScreen("04 - Puesta en marcha", 0)
   Button "Botón_3" at 2,433 size 160x47; TextOff 'Estado'
      on Click: ActivateScreen("02 - Estado", 0)

screen "03 - Registro alarmas" 800x480, template "Plantilla_1"
   Button "Botón_1" at 161,431 size 160x48; TextOff 'Estado'
      on Click: ActivateScreen("02 - Estado", 0)
   TextField "Campo de texto_5" at 286,300 size 16x23; Text 'Text'
   Button "Botón_3" at 321,431 size 161x48; TextOff 'Reset'
      on Click: SetBit("Reset"); ResetBit("HomingOk"); ResetBit("Marcha")
      Appearance <- "Alarma_ON"
   Button "Botón_4" at 640,431 size 159x48; TextOff 'Protegido'; Authorization "Administración de usuarios"
      on Click: ActivateScreen("04 - Puesta en marcha", 0)
   AlarmView "Visor de avisos_1" at 0,28 size 799x404
   Button "Botón_2" at 0,432 size 161x47; TextOff 'Homing'
      on Click: ActivateScreen("01 - Pantalla_Inicializacion", 0)
      Visibility <- "Marcha"
   Button "Botón_5" at 1,432 size 161x47; TextOff 'Homing'
      Visibility <- "Marcha"

screen "04 - Puesta en marcha" 800x480, template "Plantilla_1"
   IOField "Campo ES_1" at 66,114 size 101x53; FormatPattern s999999999.999
      ProcessValue <- "PM_MovX"
   IOField "Campo ES_2" at 66,186 size 101x53; FormatPattern s999999999.999
      ProcessValue <- "PM_MovY"
   IOField "Campo ES_3" at 66,258 size 101x53; FormatPattern s9999999999
      ProcessValue <- "PM_TChFull"
   TextField "Campo de texto_1" at 193,129 size 141x23; Text 'Movimiento en X'
   TextField "Campo de texto_2" at 193,197 size 141x23; Text 'Movimiento en Y'
   TextField "Campo de texto_3" at 193,265 size 286x23; Text 'Tiempo de espera para canal lleno'
   Button "Botón_1" at 199,431 size 99x48; TextOff 'Est'
      on Click: ActivateScreen("02 - Estado", 0)

Template "Plantilla_1" 800x480
   DateTimeField "Plantilla_Campo de fecha y hora_1" at 596,2 size 197x24
   GraphicView "Plantilla_Visor de gráficos_1" at 9,2 size 76x24; Picture "eProC Logo Paneles Parte B"
*)